(* CODESYS project AI3to1.20210303.1.project

Project tree, tasks and I/O mapping:
  Device : Changsha Xiangji-ARM Cortex A9(xilinx zynq7000)-linux, Changsha Xiangji Hiden Technology Co.Ltd, version 3.5.10.40
    application Application
      libraries: Standard, * (System); SysFile, 3.5.15.0 (System); SysTypes2 Interfaces, * (System); SysShm, * (System); CAA Mathematics, * (CAA Technical Workgroup); SysTime, 3.5.9.0 (System); VisuDialogs, * (System); CAA Types Extern, * (CAA Technical Workgroup); CAA SerialCom, * (CAA Technical Workgroup); SysMem, * (System); CAA File, * (CAA Technical Workgroup); Util, * (System); CAA DTUtil Extern, * (CAA Technical Workgroup); CAA Storage, 3.5.13.0 (CAA Technical Workgroup); CAA Net Base Services, 3.5.15.0 (CAA Technical Workgroup); CAA Memory, 3.5.12.0 (CAA Technical Workgroup)
      task c_MainTask (cyclic, interval 20 ms, priority 20) calls prg_ai3to1
      fbs/
        function block AI3to1 [ST]: is_moved
      programs/
        program prg_ai3to1 [CFC]
      trace Trace (task c_MainTask): prg_ai3to1.AI_01, prg_ai3to1.AI_02, prg_ai3to1.ai3to1_01.ai_out, prg_ai3to1.AI_03
    IoDrvMIC7001 : IoDrvMIC7001, Cyber-MI, version 19.1.1
        input  Application.prg_ai3to1.AI_02 : DWORD  // Ai09@D18
        input  Application.prg_ai3to1.AI_03 : DWORD  // Ai10@D20
        input  Application.prg_ai3to1.AI_01 : DWORD  // Ai17@D16
        output hb_do_L : BOOL  // Do24-Ai42@C23
        output hb_do_R : BOOL  // Do25-Ai43@C35
        output hb_pwm_L : DWORD  // PWM00@C25
        output hb_pwm_R : DWORD  // PWM01@C24
        unmapped channels: Ai00@C16, Ai01@C28, Ai02@C17, Ai03@C29, Ai04@C30, Ai05@C19, Ai06@C31, Ai07@C20, Ai08@C18, Ai11@D31, Ai12@D19, Ai13@D30, Ai14@D29, Ai15@D17, Ai16@D28, Ai18-Do00@C25, Ai19-Do01@C24, Ai20-Do02@C13, Ai21-Do03@C01, Ai22-Do04@C03, Ai23-Do05@C04, Ai24-Do06@C05, Ai25-Do07@C06, Ai26-Do08@C08, Ai27-Do09@C09, Ai28-Do10@C10, Ai29-Do11@C11, Ai30-Do12@D34, Ai31-Do13@D35, Ai32-Do14@D23, Ai33-Do15@D12, Ai34-Do16@D10, Ai35-Do17@D09, Ai36-Do18@D08, Ai37-Do19@D07, Ai38-Do20@D05, Ai39-Do21@D04, Ai40-Do22@D03, Ai41-Do23@D02, Ai42-Do24@C23,
          Ai43-Do25@C35, Ai44-Do26@D24, Ai45-Do27@D13, Ai46-Ao00@C22, Ai47-Ao01@D14, %ID86 Ai48_Pi02, Ai49_Out5V, Ai50_VCC, Ai51_VCC_L, Ai52_VCC_R, Ai53_Pwm-i0, Ai54_Pwm-i1, Ai55_Pwm-i2, Ai56_Pwm-i3, Ai57_CPU-T, Ai58_G-x, Ai59_G-y, Ai60_G-z, Ai61-reserved, Ai62-IO-cntr, Ai63-CDS-cntr, Di00-Ai00@C16, Di01-Ai01@C28, Di02-Ai02@C17, Di03-Ai03@C29, Di04-Ai04@C30, Di05-Ai05@C19, Di06-Ai06@C31, Di07-Ai07@C20, Di08-Ai08@C18, Di09-Ai09@D18, Di10-Ai10@D20, Di11-Ai11@D31, Di12-Ai12@D19, Di13-Ai13@D30, Di14-Ai14@D29, Di15-Ai15@D17, Di16-Ai16@D28, Di17-Ai17@D16, Di18-Ai18@C25,
          Di19-Ai19@C24, Di20-Ai20@C13, Di21-Ai21@C01, Di22-Ai22@C03, Di23-Ai23@C04, Di24-Ai24@C05, Di25-Ai25@C06, Di26-Ai26@C08, Di27-Ai27@C09, Di28-Ai28@C10, Di29-Ai29@C11, Di30-Ai30@D34, Di31-Ai31@D35, Di32-Ai32@D23, Di33-Ai33@D12, Di34-Ai34@D10, Di35-Ai35@D09, Di36-Ai36@D08, Di37-Ai37@D07, Di38-Ai38@D05, Di39-Ai39@D04, Di40-Ai40@D03, Di41-Ai41@D02, Di42-Ai42@C23, Di43-Ai43@C35, Di44-Ai44@D24, Di45-Ai45@D13, Di46-Ai46@C22, Di47-Ai47@D14, Di48-Pi00@C15, Di49-Pi01@C14, Di50-Pi02@D22, Di51-Pi03@D21, Di52-reserved, Di53-reserved, Di54-reserved, Di55-reserved, Di56-reserved, Di57-reserved, Di58-reserved,
          Di59-reserved, Di60-reserved, Di61-reserved, Di62-reserved, Di63-reserved, Pi00-Di48@C15, Pi01-Di49@C14, Pi02-Di50@D22, Pi03-Di51@D21, Do00-Ai18@C25, Do01-Ai19@C24, Do02-Ai20@C13, Do03-Ai21@C01, Do04-Ai22@C03, Do05-Ai23@C04, Do06-Ai24@C05, Do07-Ai25@C06, Do08-Ai26@C08, Do09-Ai27@C09, Do10-Ai28@C10, Do11-Ai29@C11, Do12-Ai30@D34, Do13-Ai31@D35, Do14-Ai32@D23, Do15-Ai33@D12, Do16-Ai34@D10, Do17-Ai35@D09, Do18-Ai36@D08, Do19-Ai37@D07, Do20-Ai38@D05, Do21-Ai39@D04, Do22-Ai40@D03, Do23-Ai41@D02, Do26-Ai44@D24, Do27-Ai45@D13, Do28-Pwmi00@C33, Do29-Pwmi01@C34, Do30-Pwmi02@D25, Do31-Pwmi03@D26, PWM02@C13,
          PWM03@C01, PWM04@C03, PWM05@C04, PWM06@C05, PWM07@C06, PWM08@C08, PWM09@C09, PWM10@C10, PWM11@C11, PWM12@D34, PWM13@D35, PWM14@D23, PWM15@D12, PWM16@D10, PWM17@D09, PWM18@D08, PWM19@D07, PWM20@D05, PWM21@D04, PWM22@D03, PWM23@D02, PWM24@C23, PWM25@C35, PWM26@D24, PWM27@D13, PWM28-Pwmi00@C33, PWM29-Pwmi01@C34, PWM30-Pwmi02@D25, PWM31-Pwmi03@D26, PWM_I_0@C33, PWM_I_1@C34, PWM_I_2@D25, PWM_I_3@D26, Ao00-Ai46@C22, Ao01-Ai47@D14, LED_run, LED_err, LED_usr, ctrl_ai_raw, ctrl_adjust,
          ctrl_adj0, ctrl_adj1, ctrl_adj2, ctrl_adj3, ctrl_adj4
    SoftMotion General Axis Pool
  libraries: VisuSymbols, 3.5.10.0 (System)
  5ce3da45-db07-42e7-a21c-a00fff4ed8f6|C:\Users\zhou\p01.bmp
  5ce3da45-db07-42e7-a21c-a00fff4ed8f6|C:\working\p01.bmp
  5ce3da45-db07-42e7-a21c-a00fff4ed8f6|台达驱动器.jpg
  5ce3da45-db07-42e7-a21c-a00fff4ed8f6|C:\working\file.bmp
  text list GlobalTextList
  5ce3da45-db07-42e7-a21c-a00fff4ed8f6|mir3501.jpg
  text list System
  5ce3da45-db07-42e7-a21c-a00fff4ed8f6|delta.jpg
*)

// Device/Application/programs/prg_ai3to1
PROGRAM prg_ai3to1
VAR
	ai3to1_01:ai3to1;
	AI_01:DWORD;
	AI_02:DWORD;
	AI_03:DWORD;
END_VAR
//

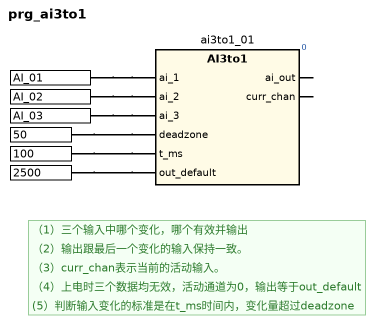
// （1）三个输入中哪个变化，哪个有效并输出
// （2）输出跟最后一个变化的输入保持一致。
// （3）curr_chan表示当前的活动输入。
// （4）上电时三个数据均无效，活动通道为0，输出等于out_default
// (5）判断输入变化的标准是在t_ms时间内，变化量超过deadzone
ai3to1_01(ai_1 := AI_01, ai_2 := AI_02, ai_3 := AI_03, deadzone := 50, t_ms := 100, out_default := 2500); // AI3to1

END_PROGRAM

// Device/Application/fbs/AI3to1
FUNCTION_BLOCK AI3to1
VAR_INPUT
	ai_1 : DWORD := 0;
	ai_2 : DWORD := 0;
	ai_3 : DWORD := 0;
	deadzone : DINT := 15;  // AI 变化死区值
	t_ms : DINT := 100;     // 功能块运行时间间隔（毫秒）
	out_default :DWORD := 0;  // 输出默认值
END_VAR

VAR_OUTPUT
	ai_out : DWORD := 0;
	curr_chan :DINT := 0;  // 当前活动通道的编号
END_VAR
VAR
	stat : DINT := 0;
	ai_old_1 : DWORD;
	ai_old_2 : DWORD;
	ai_old_3 : DWORD;
	tick:ton;

END_VAR


tick(in := NOT tick.Q, pt := ANY_TO_TIME(t_ms));
IF NOT tick.Q THEN
	RETURN;
END_IF


CASE stat OF
0:
    stat := 5;
	ai_out := out_default;
	curr_chan := 0;
10:
	ai_out := ai_1;	
20:
    ai_out := ai_2;
30:
    ai_out := ai_3;
END_CASE

IF is_moved(1) THEN
	curr_chan := 1;
	stat := 10;
ELSIF is_moved(2) THEN
	curr_chan := 2;
	stat := 20;
ELSIF is_moved(3) THEN
	curr_chan := 3;
	stat := 30;
END_IF

METHOD is_moved : BOOL
VAR_INPUT
	index:DINT;
END_VAR

VAR
	ai:DWORD := 0;
	old:DWORD := 0;
END_VAR
CASE index OF
1:
    ai := ai_1;
	old := ai_old_1;
	ai_old_1 := ai_1;
2:
    ai := ai_2;
	old := ai_old_2;
	ai_old_2 := ai_2;
3:
    ai := ai_3;
	old := ai_old_3;
	ai_old_3 := ai_3;
END_CASE

IF ABS(ANY_TO_DINT(ai) - ANY_TO_DINT(old)) > deadzone THEN
	is_moved := TRUE;
ELSE
	is_moved := FALSE;
END_IF

IF old = 0 THEN
	is_moved := FALSE;
END_IF
END_METHOD

END_FUNCTION_BLOCK

(* text list System (id | default)
  Apr | Apr
  April | April
  Aug | Aug
  August | August
  Dec | Dec
  December | December
  Feb | Feb
  February | February
  Fri | Fri
  Friday | Friday
  Jan | Jan
  January | January
  Jul | Jul
  July | July
  Jun | Jun
  June | June
  Mar | Mar
  March | March
  May | May
  May_3Letter | May
  Mon | Mon
  Monday | Monday
  Nov | Nov
  November | November
  Oct | Oct
  October | October
  Sat | Sat
  Saturday | Saturday
  Sep | Sep
  September | September
  Sun | Sun
  Sunday | Sunday
  Thu | Thu
  Thursday | Thursday
  Tue | Tue
  Tuesday | Tuesday
  Wed | Wed
  Wednesday | Wednesday
   |  *)
